(* IEC 61131-3 sources: programs/VI-54/VI-54_20171205/VI-54_20171205/Stations/PLC_VI54/VI-54_171014/Class/Vi54_Control, 1 file *)

(* ---- Vi54_Control.st ---- *)
(*!
<Class
	Name               = "Vi54_Control"
	Revision           = "0.0"
	RealtimeTask       = "true"
	CyclicTask         = "true"
	BackgroundTask     = "false"
	Sigmatek           = "false"
	OSInterface        = "false"
	HighPriority       = "false"
	Automatic          = "false"
	UpdateMode         = "Prescan"
	SharedCommandTable = "true"
	Objectsize         = "(780,1020)">
	<Channels>
		<Server Name="__________" Visualized="false" Initialize="false" WriteProtected="true" Retentive="false"/>
		<Server Name="CleaningJog" Visualized="true" Initialize="false" WriteProtected="false" Retentive="false"/>
		<Server Name="CleaningJogDistance" Visualized="true" Initialize="false" WriteProtected="false" Retentive="File"/>
		<Server Name="CleaningJogOption" Visualized="true" Initialize="false" WriteProtected="false" Retentive="File"/>
		<Server Name="CleaningMode" Visualized="true" Initialize="false" WriteProtected="false" Retentive="false"/>
		<Server Name="CleaningSpeed" Visualized="true" Initialize="false" WriteProtected="false" Retentive="File"/>
		<Server Name="CPU_Load" Visualized="true" Initialize="false" WriteProtected="true" Retentive="false"/>
		<Server Name="ExternalPause" Visualized="true" Initialize="false" WriteProtected="true" Retentive="false"/>
		<Server Name="Gestart" Visualized="true" Initialize="false" WriteProtected="true" Retentive="false"/>
		<Server Name="Gestopt" Visualized="true" Initialize="false" WriteProtected="true" Retentive="false"/>
		<Server Name="InternalPause" Visualized="true" Initialize="false" WriteProtected="true" Retentive="false"/>
		<Server Name="JogButtonVisual" Visualized="true" Initialize="false" WriteProtected="true" Retentive="false"/>
		<Server Name="MasterOverrule" Visualized="true" Initialize="false" WriteProtected="false" Retentive="false"/>
		<Server Name="PauseActive" Visualized="true" Initialize="false" WriteProtected="false" Retentive="File"/>
		<Server Name="PauseDelay" Visualized="true" Initialize="false" WriteProtected="false" Retentive="File"/>
		<Server Name="PauseSignalOptions" Visualized="true" Initialize="false" WriteProtected="false" Retentive="File"/>
		<Server Name="Reset" Visualized="true" Initialize="false" WriteProtected="false" Retentive="false"/>
		<Server Name="ResetKnopVisual" Visualized="true" Initialize="false" WriteProtected="true" Retentive="false"/>
		<Server Name="RunState" Visualized="true" Initialize="false" WriteProtected="true" Retentive="false"/>
		<Server Name="RunStateInfeedConv" Visualized="true" Initialize="false" WriteProtected="true" Retentive="false"/>
		<Server Name="UseInpAnalogeSpeed" Visualized="true" Initialize="false" WriteProtected="false" Retentive="File"/>
		<Client Name="ClaxonComm" Required="true" Internal="false"/>
		<Client Name="Comm_CameraMaster" Required="true" Internal="false"/>
		<Client Name="Comm_Conveyors" Required="true" Internal="false"/>
		<Client Name="Comm_Xaxles" Required="true" Internal="false"/>
		<Client Name="Comm_Yaxles" Required="true" Internal="false"/>
		<Client Name="iDrivesEnabled" Required="true" Internal="false"/>
		<Client Name="iDrivesOk" Required="true" Internal="false"/>
		<Client Name="iExternRelease" Required="true" Internal="false"/>
		<Client Name="iLineSpeed" Required="true" Internal="false"/>
		<Client Name="iSafetyOK" Required="true" Internal="false"/>
		<Client Name="iStart" Required="true" Internal="false"/>
		<Client Name="iStop" Required="true" Internal="false"/>
		<Client Name="LampComm" Required="true" Internal="false"/>
		<Client Name="MglobalData" Required="true" Internal="true"/>
		<Client Name="oMachineOK" Required="true" Internal="false"/>
		<Client Name="oPause" Required="true" Internal="false"/>
		<Client Name="oResetSignal" Required="true" Internal="false"/>
		<Client Name="Standard3" Required="true" Internal="true"/>
		<Client Name="vError" Required="true" Internal="false"/>
	</Channels>
	<Network Name="Vi54_Control">
		<!-- List of Components in this network -->
		<Components>
			<Object
				Name       = "_base"
				Class      = "RecipeBase"
				Position   = "(354,120)"
				Visualized = "false">
				<Channels>
					<Server Name="Comm"/>
					<Client Name="MainRecipe"/>
				</Channels>
			</Object>
			<Object
				Name       = "MglobalData"
				Class      = "MerkerEx"
				Position   = "(300,330)"
				Visualized = "true"
				Remotely   = "true">
				<Channels>
					<Server Name="m_udLength"/>
					<Client Name="ThreadSafe" Value="0"/>
				</Channels>
			</Object>
			<Object
				Name           = "Standard3"
				Class          = "Standard"
				Position       = "(330,480)"
				Visualized     = "false"
				BackgroundTime = "1000 ms">
				<Channels>
					<Server Name="ClassSvr"/>
				</Channels>
			</Object>
		</Components>
		<Comments>
		</Comments>
		<!-- List of Connections in this network -->
		<Connections>
			<Connection Source="this.MglobalData" Destination="MglobalData.m_udLength"/>
			<Connection Source="this.Standard3" Destination="Standard3.ClassSvr"/>
			<Connection Source="this.Comm" Destination="_base.Comm" Vertices="(938,210),(654,210),"/>
			<Connection Source="_base.MainRecipe" Destination="this.MainRecipe" Vertices="(354,210),(38,210),"/>
		</Connections>
		<!-- Headerfiles -->
		<Options>
		</Options>
	</Network>
</Class>
*)
#pragma using RecipeBase

Vi54_Control : CLASS
: RecipeBase
  //Servers:
	Gestart 	: SvrCh_DINT;
	Gestopt 	: SvrCh_DINT;
	InternalPause 	: SvrCh_DINT;
	ExternalPause 	: SvrCh_DINT;
	CPU_Load 	: SvrCh_DINT;
	Reset 	: SvrCh_DINT;
	MasterOverrule 	: SvrCh_DINT;
	CleaningMode 	: SvrCh_DINT;
	CleaningJogOption 	: SvrCh_OptiesEnum;
	CleaningJog 	: SvrCh_DINT;
	JogButtonVisual 	: SvrCh_DINT;
	CleaningSpeed 	: SvrCh_DINT;
	CleaningJogDistance 	: SvrCh_DINT;
	PauseSignalOptions 	: SvrCh_PauseFunctions;
	PauseActive 	: SvrCh_OptiesEnum;
	PauseDelay 	: SvrCh_DINT;
	ResetKnopVisual 	: SvrCh_DINT;
	UseInpAnalogeSpeed 	: SvrCh_OptiesEnum;
	__________ 	: SvrCh_DINT;
	RunState 	: SvrCh_RunningStateEnum;
	RunStateInfeedConv 	: SvrCh_RunningStateEnum;
  //Clients:
	Comm_Xaxles 	: CltChCmd_X_Axle_Correction;
	Comm_Yaxles 	: CltChCmd_Y_Axle_Correction;
	Comm_CameraMaster 	: CltChCmd_Camera_Master;
	Comm_Conveyors 	: CltChCmd_InfeedBelt;
	iLineSpeed 	: CltChCmd_SpeedInput;
	iStart 	: CltCh_DINT;
	iStop 	: CltCh_DINT;
	LampComm 	: CltChCmd_Banner_EZlight;
	ClaxonComm 	: CltChCmd_Claxon;
	iSafetyOK 	: CltCh_DINT;
	iExternRelease 	: CltCh_DINT;
	oMachineOK 	: CltCh_DINT;
	oPause 	: CltCh_DINT;
	iDrivesOk 	: CltCh_DINT;
	iDrivesEnabled 	: CltCh_DINT;
	oResetSignal 	: CltCh_DINT;
	vError 	: CltCh_DINT;
	MglobalData 	: CltChCmd_MerkerEx;
	Standard3 	: CltChCmd_Standard;
  //Variables:
		NoError 	: DINT;
		StartingUp 	: DINT;
		GlobalDataPtr 	: ^GlobalDataStr;
		PauseSignal 	: DINT;
		PauzeOverride 	: DINT;
		CalcLineSpeed 	: DINT;
		WaitForNextPausePuls 	: DINT;
		TmrPause 	: UDINT;
		PauseOverride 	: DINT;
  //Functions:

	FUNCTION VIRTUAL GLOBAL Init;

	FUNCTION VIRTUAL GLOBAL CyWork
		VAR_INPUT
			EAX 	: UDINT;
		END_VAR
		VAR_OUTPUT
			state (EAX) 	: UDINT;
		END_VAR;

	FUNCTION VIRTUAL GLOBAL RtWork
		VAR_INPUT
			EAX 	: UDINT;
		END_VAR
		VAR_OUTPUT
			state (EAX) 	: UDINT;
		END_VAR;

	FUNCTION VIRTUAL GLOBAL Background
		VAR_INPUT
			EAX 	: UDINT;
		END_VAR
		VAR_OUTPUT
			state (EAX) 	: UDINT;
		END_VAR;

	FUNCTION GLOBAL GlobalData;

	FUNCTION GLOBAL ResetComm;
  //Tables:
	FUNCTION @STD
		VAR_OUTPUT
			ret_code	: CONFSTATES;
		END_VAR;
	FUNCTION GLOBAL TAB @CT_;
END_CLASS;

#pragma using MerkerEx
#pragma using Standard
#pragma usingLtd Banner_EZlight
#pragma usingLtd Camera_Master
#pragma usingLtd Claxon
#pragma usingLtd InfeedBelt
#pragma usingLtd SpeedInput
#pragma usingLtd X_Axle_Correction
#pragma usingLtd Y_Axle_Correction

FUNCTION VIRTUAL GLOBAL Vi54_Control::Init

  if mGlobalData.GetSize() <> sizeof(GlobalDataStr) then
    mGlobalData.SetSize(udSize:= sizeof(GlobalDataStr));
  end_if;

  // open init methode of baseclass
  RecipeBase::Init();

  // Only at first scan
  if _FirstScan = 1 then
    GlobalDataPtr$^Usint := mGlobalData.GetDataPtr();

    // Set pointers
    Comm_Conveyors.InitTask(SetGlobalPtr:= GlobalDataPtr, SetRecipePtr:= ReceptPtr);
    Comm_Conveyors.SetStationNbr(Nbr:= 1);

    Comm_CameraMaster.InitTask(SetGlobalPtr:= GlobalDataPtr, SetRecipePtr:= ReceptPtr);

    Comm_Xaxles.InitTask(SetGlobalPtr:= GlobalDataPtr, SetRecipePtr:= ReceptPtr);
    Comm_Xaxles.SetStationNbr(Nbr:= 1);

    Comm_Yaxles.InitTask(SetGlobalPtr:= GlobalDataPtr, SetRecipePtr:= ReceptPtr);
    Comm_Yaxles.SetStationNbr(Nbr:= 1);
  end_if;

END_FUNCTION

FUNCTION VIRTUAL GLOBAL Vi54_Control::RtWork
	VAR_INPUT
		EAX 	: UDINT;
	END_VAR
	VAR_OUTPUT
		state (EAX) 	: UDINT;
	END_VAR

  // Open realtime tasks
  Comm_CameraMaster.RtTask();

	state := READY;

END_FUNCTION

FUNCTION VIRTUAL GLOBAL Vi54_Control::CyWork
	VAR_INPUT
		EAX 	: UDINT;
	END_VAR
	VAR_OUTPUT
		state (EAX) 	: UDINT;
	END_VAR

  // Read inputs
  iSafetyOK       := iSafetyOK.Read();
  iDrivesOk       := iDrivesOk.Read();
  iDrivesEnabled  := iDrivesEnabled.Read();
  iStart          := iStart.Read();
  iStop           := iStop.Read();
  CPU_Load        := _CPULOAD;

  // Open methodes
  Comm_CameraMaster.CyTask();
  Comm_Xaxles.CyTask();
  Comm_Yaxles.CyTask();
  Comm_Conveyors.CyTask();
  GlobalData();
  ResetComm();

  // Calculate the actual line speed
  if UseInpAnalogeSpeed = Actief then
    iLineSpeed.MyRtTask(InputSetting:= SpeedInput::eInput::eAnalog);
    CalcLineSpeed := to_dint(to_real iLineSpeed.ActInfeedSpeed ToMMperSec);
  else
    CalcLineSpeed := to_dint(to_real ReceptPtr^.Machine.LineSpeed ToMMperSec);
  end_if;

  // Cleaning jog function
  JogButtonVisual$dint := (CleaningMode = 1 & CleaningJogOption = Actief);
  if CleaningJog = 1 then
    CleaningJog := 0;
  end_if;

   // check errors..
  if IsClientConnected(#vError) then
    vError := vError.Read();
  else
    vError := 0;
  end_if;
  NoError := (vError = 0);

  // ResetKnop visable
  if iSafetyOK = 0  | NoError = 0 then
    ResetKnopVisual := 1;
  else
    ResetKnopVisual := 0;
  end_if;

  // Runstatussen
  if iSafetyOK = 0 then  // NOODSTOP
    Gestart := 0;
    CleaningMode := 0;
    StartingUp := 0;
    RunState := eNoodstopStatus;
  elsif NoError = 0 then // storing
    Gestart := 0;
    CleaningMode := 0;
    StartingUp := 0;
    RunState := eErrorStatus;
  elsif iStop = 0 & (Gestart = 1 | CleaningMode = 1) then // stop knop
    Gestart := 0;
    CleaningMode := 0;
    if NoError = 0 then  // met stop knop ook reset mogelijk !!
      oResetSignal := 1;
    end_if;
    RunState := eStopStatus;
  elsif CleaningMode = 1 & Gestart = 0 then  // machine in schoonmaak stand
    Gestart := 0;
    RunState := eCleaningStatus;
  elsif iStart = 1 & Gestart = 0 then
    CleaningMode := 0;
    Gestart := 1;
  else
    if StartingUp = 1 then
      Gestart := 0;
      if GlobalDataPtr^.gMachineData.Reference_Amount = GlobalDataPtr^.gMachineData.Act_Reference_Amount then
        StartingUp := 0;
      end_if;
    elsif Gestart = 1 then
      if GlobalDataPtr^.gMachineData.Reference_Amount <> GlobalDataPtr^.gMachineData.Act_Reference_Amount then
        Gestart := 0;  // na opstarten opnieuw start geven..
        StartingUp := 1;
        RunState := eStartUpStatus;
      end_if;
      if StartingUp = 0 & PauseSignal = 1 then
        CleaningMode := 0;
        RunState := eRunStatus;
      elsif StartingUp = 0 & PauseSignal = 0 then
        CleaningMode := 0;
        Runstate := ePauseStatus;
      end_if;
    else
      RunState := eStopStatus;
    end_if;
  end_if;
  Gestopt := (Gestart = 0);

  // Pauze signaal, verschillende keuzes betreft inlezen
  if PauseActive = actief then
    iExternRelease  := iExternRelease.Read();
    if PauseSignalOptions = NormalyClosed then // normaly closed
      if iExternRelease = 0 then
        PauseSignal := 0;
      else
        PauseSignal := 1;
      end_if;
    elsif PauseSignalOptions = NormalyOpen then // normaly open
      if iExternRelease = 1 then
        PauseSignal := 0;
      else
        PauseSignal := 1;
      end_if;
    elsif PauseSignalOptions = Puls then // Met een puls pause signaal in- en uitschakelen
      if Standard3.R_TRIG(CLK:= iExternRelease) then
        WaitForNextPausePuls := 1;
        PauseSignal := 0;
      elsif WaitForNextPausePuls = 1 & Standard3.R_TRIG(CLK:= iExternRelease) then
        WaitForNextPausePuls := 0;
        PauseSignal := 1;
      end_if;
    end_if;

    if PauseSignal = 0 & CleaningMode = 0 then // hef op bij schoonmaken
      if (ops.tAbsolute - TmrPause) >= to_udint(PauseDelay * _100MS) then // vertraagd stop signaal (Vi-08)
        PauseOverride := 0;
      end_if;
    else
      PauseOverride := 1000;
      TmrPause := Ops.tAbsolute;
    end_if;
  else
    PauseSignal := 1;
    PauseOverride := 1000;
    TmrPause := Ops.tAbsolute;
  end_if;

  if IsClientConnected(#oPause) then
    oPause := (PauseSignal = 1 & RunState = eRunStatus);
    oPause.Write (oPause);
  end_if;

  // Leds from the piëzo buttons
  if NoError = 0 then
    iStart := -1;
  elsif StartingUp = 1 then
    iStart := -2;
  elsif Gestart = 0 then
    iStart := 0;
  elsif (PauseSignal = 0 & PauseActive = actief) then
    iStart := -3;
  else
    iStart := 1;
  end_if;
  iStart.Write(input:=iStart);

  // Set light collors
  if Runstate = eRunStatus then
    LampComm.LightCollors(iCollor:= Banner_EZlight::eGreenOn);
  elsif Runstate = ePauseStatus then
    LampComm.LightCollors(iCollor:= Banner_EZlight::eGreenFlashing);
  elsif Runstate = eStopStatus then
    LampComm.LightCollors(iCollor:= Banner_EZlight::eWhiteOn);
  elsif Runstate = eNoodstopStatus then
    LampComm.LightCollors(iCollor:= Banner_EZlight::eRedOn);
  elsif Runstate = eErrorStatus then
    LampComm.LightCollors(iCollor:= Banner_EZlight::eYellowOn);
  end_if;

  // Set claxon sound
  if ClaxonComm.ClaxonActief = Actief then
    if Runstate = eNoodstopStatus | Runstate = eErrorStatus then
      ClaxonComm.ClaxonState(State:= 1);
    else
      ClaxonComm.ClaxonState(State:= 0);
    end_if;
  end_if;

	state := READY;

END_FUNCTION

FUNCTION VIRTUAL GLOBAL Vi54_Control::Background
	VAR_INPUT
		EAX 	: UDINT;
	END_VAR
	VAR_OUTPUT
		state (EAX) 	: UDINT;
	END_VAR

  // Open Background methodes

	state := READY;

END_FUNCTION

FUNCTION GLOBAL Vi54_Control::ResetComm

  if Reset = 1 then
    Comm_CameraMaster.ResetErrors();
    Comm_Xaxles.ResetErrors();
    Comm_Yaxles.ResetErrors();
    Comm_Conveyors.ResetErrors();
    oResetSignal := 1;
  else
    oResetSignal := 0;
    Reset        := 0;
  end_if;

  oResetSignal.Write(input:= oResetSignal);

END_FUNCTION

FUNCTION GLOBAL Vi54_Control::GlobalData

  // global data pointers vullen
  GlobalDataPtr^.gRunStatus.gRunStatusGlob               := RunState;
  GlobalDataPtr^.gGeneralData.LineSpeed                  := CalcLineSpeed;
  GlobalDataPtr^.gGeneralData.iDrivesOK                  := iDrivesOk;
  GlobalDataPtr^.gGeneralData.iDrivesEnabled             := iDrivesEnabled;
  GlobalDataPtr^.gGeneralData.iNoodstopOk                := iSafetyOK;
  GlobalDataPtr^.gGeneralData.iExternrelease             := PauseSignal;
  GlobalDataPtr^.gGeneralData.PauzeOverride              := PauzeOverride;
  GlobalDataPtr^.gGeneralData.NoError                    := NoError;

  // Cleaning Settings
  GlobalDataPtr^.gGeneralData.CleaningMode               := CleaningMode;
  GlobalDataPtr^.gGeneralData.CleaningJogOption          := CleaningJogOption;
  GlobalDataPtr^.gGeneralData.CleaningJog                := CleaningJog;
  GlobalDataPtr^.gGeneralData.CleaningJogDistance        := CleaningJogDistance;
  GlobalDataPtr^.gGeneralData.CleaningSpeed              := to_dint(to_real CleaningSpeed ToMMperSec);
  GlobalDataPtr^.gGeneralData.CleaningAccDec             := to_dint(to_real 30 ToMMperSec2);

  GlobalDataPtr^.gGeneralData.oResetSignal               := oResetSignal;
  GlobalDataPtr^.gGeneralData.oMachineOK                 := oMachineOK;

  // Set runstates
  RunStateInfeedConv  := GlobalDataPtr^.gRunStatus.gRunStatusInfeedConv;

END_FUNCTION
